// SIMATIC S7-200 SMART project (STEP 7-Micro/WIN SMART), CPU ST20

SYMBOL_TABLE System Symbols
Always_On        SM0.0    // Always ON
First_Scan_On    SM0.1    // ON for the first scan cycle only
HSC0_Ctrl        SMB37    // Configure and control HSC0
HSC0_CV          SMD38    // HSC0 new current value
HSC0_PV          SMD42    // HSC0 new preset value
END_SYMBOL_TABLE

ORGANIZATION_BLOCK MAIN:OB1
TITLE=Program Comments
BEGIN
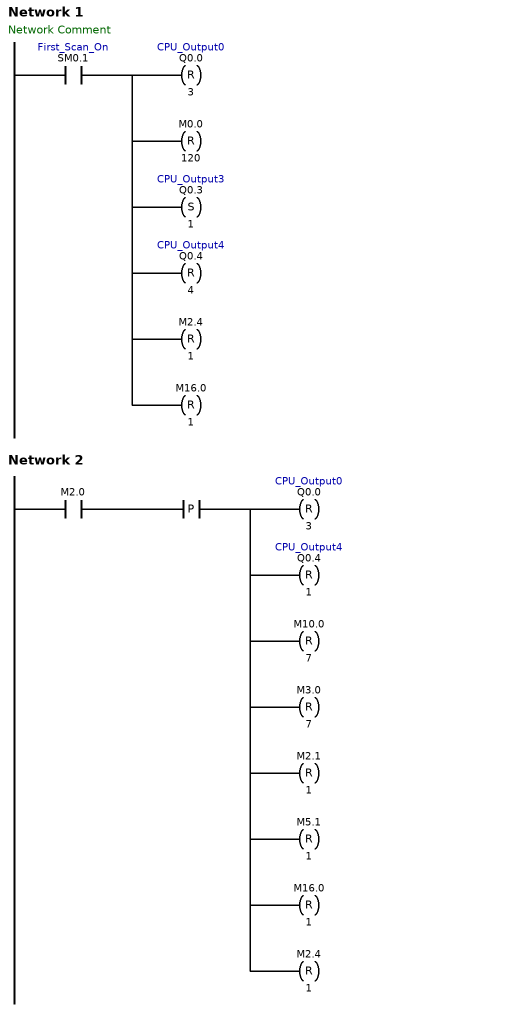
Network 1
// Network Comment
LD     First_Scan_On:SM0.1
R      CPU_Output0:Q0.0, 3
R      M0.0, 120
S      CPU_Output3:Q0.3, 1
R      CPU_Output4:Q0.4, 4
R      M2.4, 1
R      M16.0, 1
Network 2
LD     M2.0
EU
R      CPU_Output0:Q0.0, 3
R      CPU_Output4:Q0.4, 1
R      M10.0, 7
R      M3.0, 7
R      M2.1, 1
R      M5.1, 1
R      M16.0, 1
R      M2.4, 1
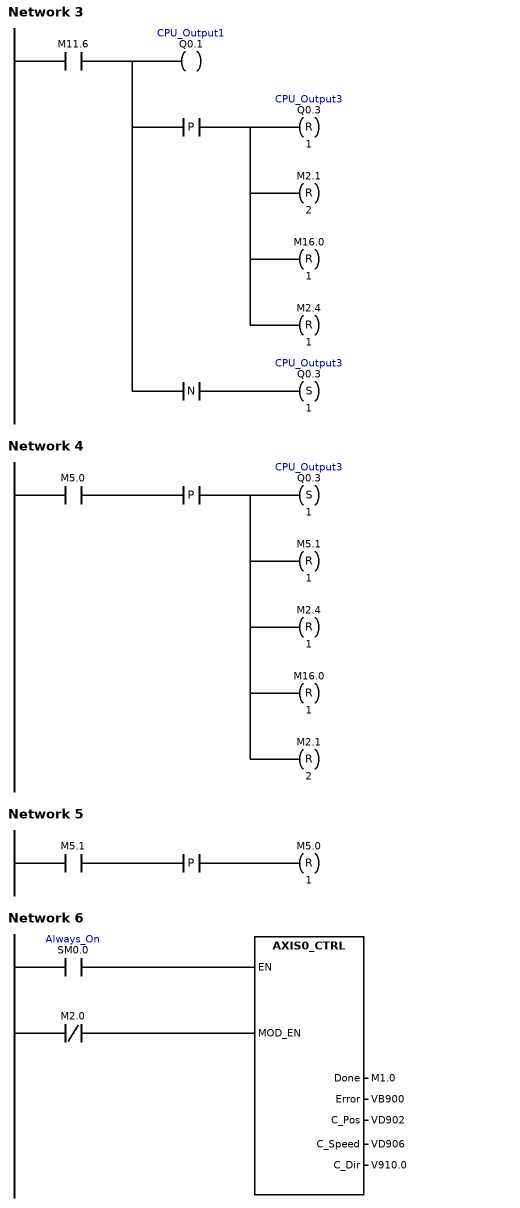
Network 3
LD     M11.6
LPS
=      CPU_Output1:Q0.1
EU
R      CPU_Output3:Q0.3, 1
R      M2.1, 2
R      M16.0, 1
R      M2.4, 1
LPP
ED
S      CPU_Output3:Q0.3, 1
Network 4
LD     M5.0
EU
S      CPU_Output3:Q0.3, 1
R      M5.1, 1
R      M2.4, 1
R      M16.0, 1
R      M2.1, 2
Network 5
LD     M5.1
EU
R      M5.0, 1
Network 6
LD     Always_On:SM0.0
=      L60.0
LDN    M2.0
=      L63.7
LD     L60.0
CALL   AXIS0_CTRL:SBR1, L63.7, M1.0, VB900, VD902, VD906, V910.0
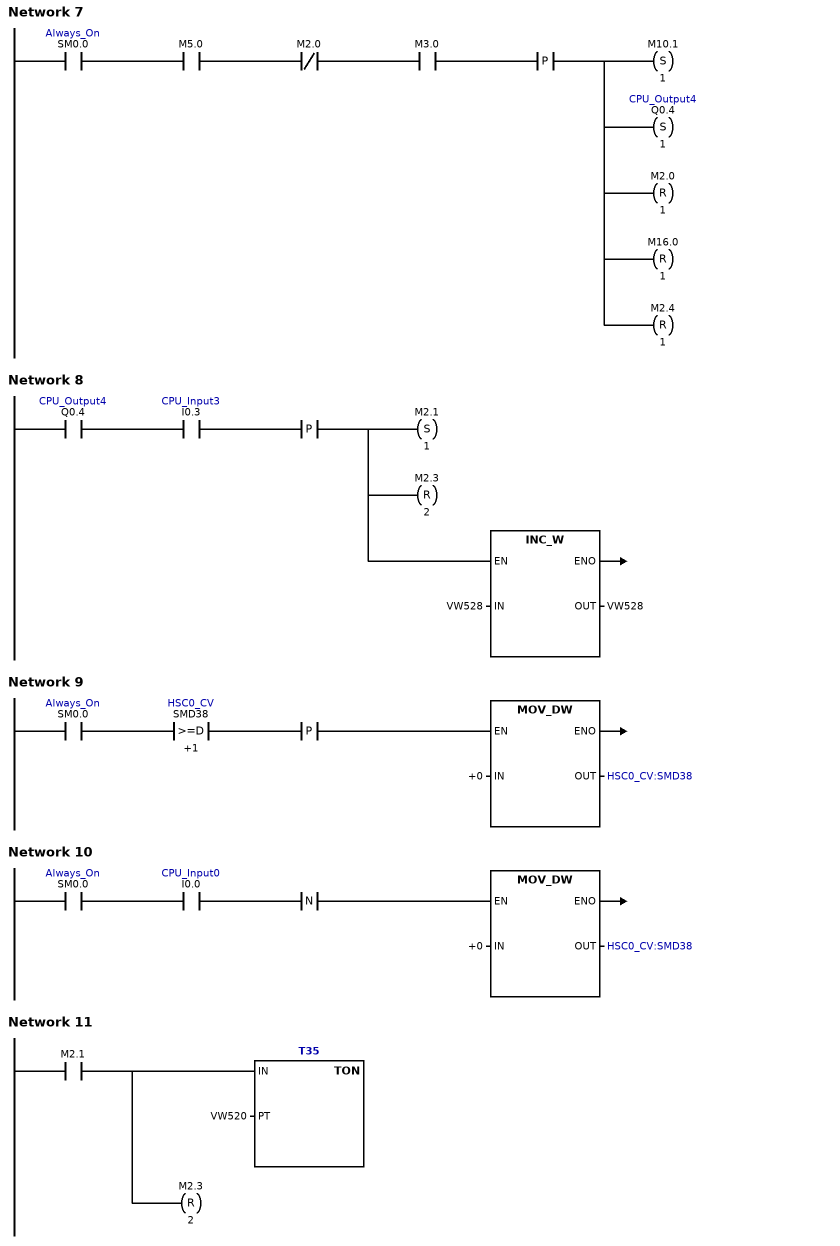
Network 7
LD     Always_On:SM0.0
A      M5.0
AN     M2.0
A      M3.0
EU
S      M10.1, 1
S      CPU_Output4:Q0.4, 1
R      M2.0, 1
R      M16.0, 1
R      M2.4, 1
Network 8
LD     CPU_Output4:Q0.4
A      CPU_Input3:I0.3
EU
S      M2.1, 1
R      M2.3, 2
INCW   VW528
Network 9
LD     Always_On:SM0.0
AD>=   HSC0_CV:SMD38, +1
EU
MOVD   +0, HSC0_CV:SMD38
Network 10
LD     Always_On:SM0.0
A      CPU_Input0:I0.0
ED
MOVD   +0, HSC0_CV:SMD38
Network 11
LD     M2.1
TON    T35, VW520
R      M2.3, 2
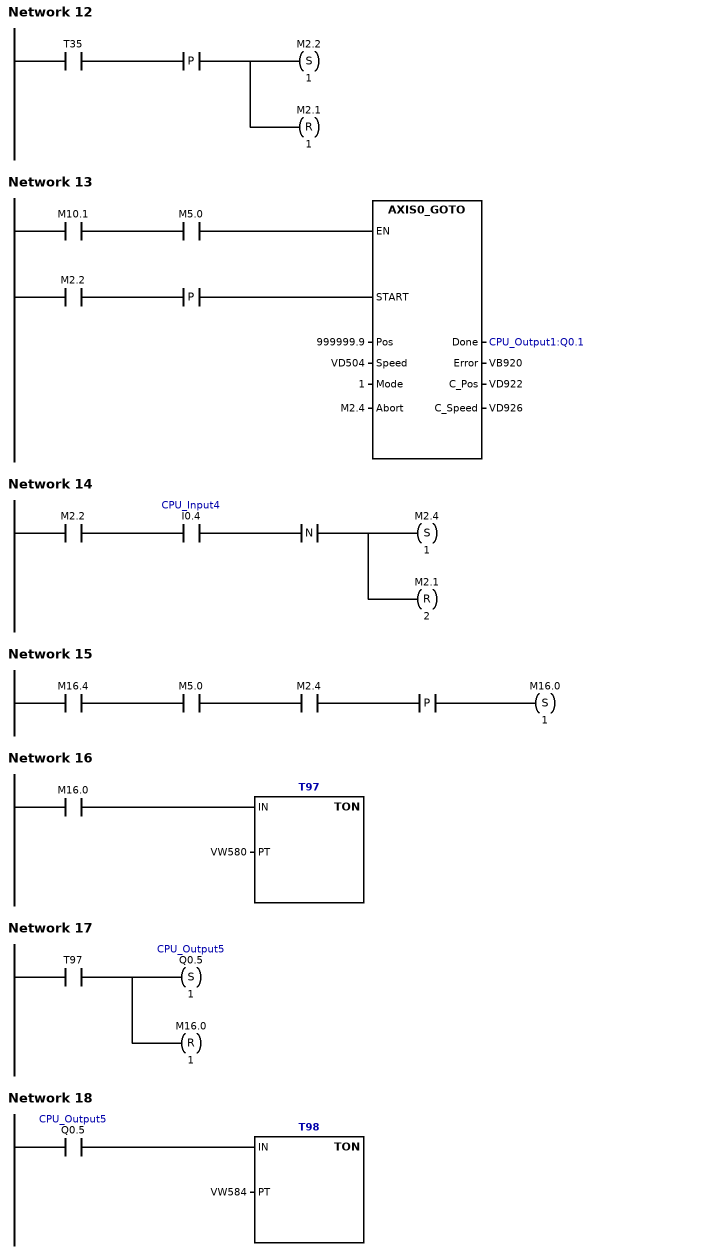
Network 12
LD     T35
EU
S      M2.2, 1
R      M2.1, 1
Network 13
LD     M10.1
A      M5.0
=      L60.0
LD     M2.2
EU
=      L63.7
LD     L60.0
CALL   AXIS0_GOTO:SBR3, L63.7, 999999.9, VD504, 1, M2.4, CPU_Output1:Q0.1, VB920, VD922, VD926
Network 14
LD     M2.2
A      CPU_Input4:I0.4
ED
S      M2.4, 1
R      M2.1, 2
Network 15
LD     M16.4
A      M5.0
A      M2.4
EU
S      M16.0, 1
Network 16
LD     M16.0
TON    T97, VW580
Network 17
LD     T97
S      CPU_Output5:Q0.5, 1
R      M16.0, 1
Network 18
LD     CPU_Output5:Q0.5
TON    T98, VW584
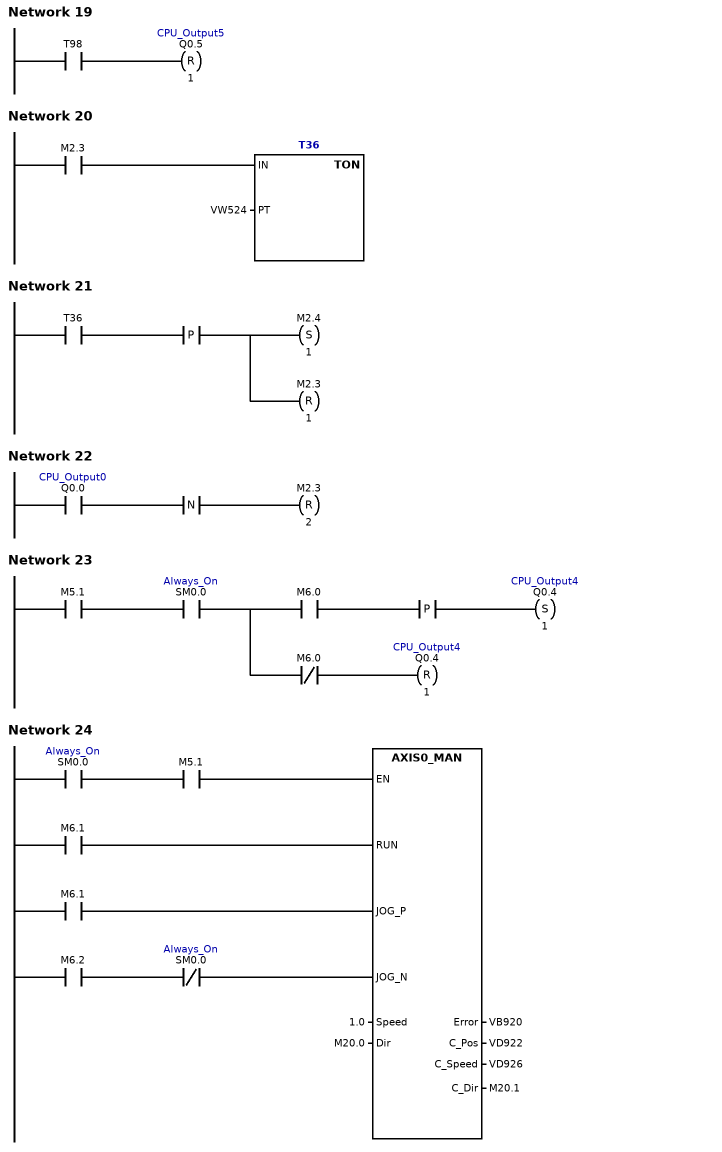
Network 19
LD     T98
R      CPU_Output5:Q0.5, 1
Network 20
LD     M2.3
TON    T36, VW524
Network 21
LD     T36
EU
S      M2.4, 1
R      M2.3, 1
Network 22
LD     CPU_Output0:Q0.0
ED
R      M2.3, 2
Network 23
LD     M5.1
A      Always_On:SM0.0
LPS
A      M6.0
EU
S      CPU_Output4:Q0.4, 1
LPP
AN     M6.0
R      CPU_Output4:Q0.4, 1
Network 24
LD     Always_On:SM0.0
A      M5.1
=      L60.0
LD     M6.1
=      L63.7
LD     M6.1
=      L63.6
LD     M6.2
AN     Always_On:SM0.0
=      L63.5
LD     L60.0
CALL   AXIS0_MAN:SBR2, L63.7, L63.6, L63.5, 1.0, M20.0, VB920, VD922, VD926, M20.1
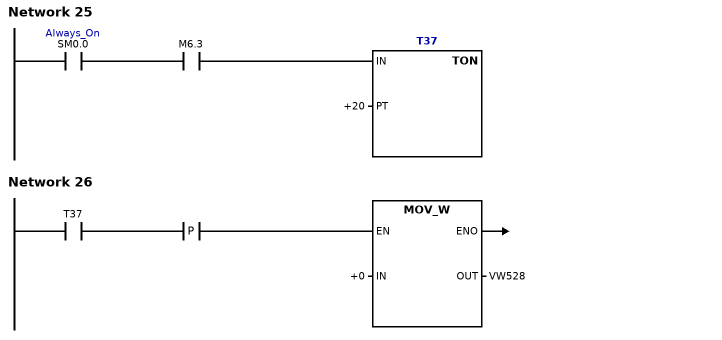
Network 25
LD     Always_On:SM0.0
A      M6.3
TON    T37, +20
Network 26
LD     T37
EU
MOVW   +0, VW528
END_ORGANIZATION_BLOCK

// SBR1: protected block, not included

// SBR2: protected block, not included

// SBR3: protected block, not included

// SBR4: protected block, not included

// SBR5: protected block, not included

// SBR6: protected block, not included

// SBR7: protected block, not included

// SBR8: protected block, not included

// SBR9: protected block, not included

// SBR10: protected block, not included

// SBR11: protected block, not included

SUBROUTINE_BLOCK HSC0_INIT_1:SBR14
TITLE=
BEGIN
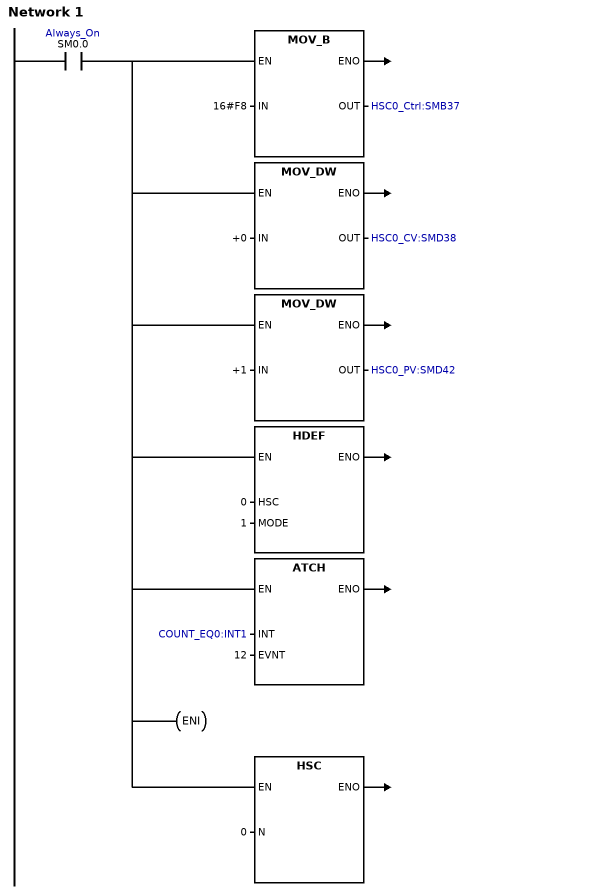
Network 1
LD     Always_On:SM0.0
MOVB   16#F8, HSC0_Ctrl:SMB37
MOVD   +0, HSC0_CV:SMD38
MOVD   +1, HSC0_PV:SMD42
HDEF   0, 1
ATCH   COUNT_EQ0:INT1, 12
ENI
HSC    0
END_SUBROUTINE_BLOCK

INTERRUPT_BLOCK COUNT_EQ0:INT1
TITLE=
BEGIN
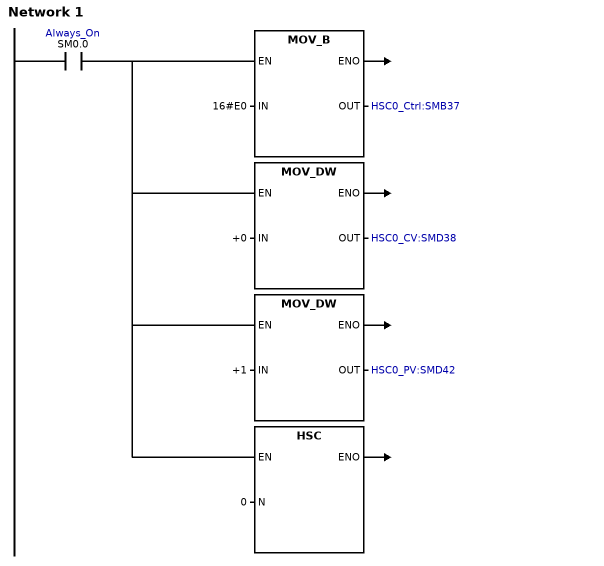
Network 1
LD     Always_On:SM0.0
MOVB   16#E0, HSC0_Ctrl:SMB37
MOVD   +0, HSC0_CV:SMD38
MOVD   +1, HSC0_PV:SMD42
HSC    0
END_INTERRUPT_BLOCK

DATA_BLOCK_TAB _PLC_DATA_1
BEGIN
VB504    16#40
VB505    16#C
VB506    16#CC
VB507    16#CD
VB529    16#38
VB581    16#A
VB585    16#A
VB900    16#82
VB902    16#43
VB903    16#4A
VB904    16#D8
VB905    16#52
VB920    16#1
VB922    16#43
VB923    16#4A
VB924    16#D8
VB925    16#52
END_DATA_BLOCK_TAB
